Fanuc KAREL source: kt00602.KL

PROGRAM KT00602
%STACKSIZE=65535
%PRIORITY=65535
%NOLOCKGROUP
VAR
I1 : INTEGER
I2 : INTEGER
OUT : REAL
BEGIN
I1=2
I2=3
I1=2
I2=3
OUT=I1
END KT00602
